{attribute addProperty BoxType "EL5101-0000-0001"}
{attribute addProperty Id "StatusAT %I*USINT811ValueAT %I*UINT1622LatchAT %I*UINT1623"}
{attribute addProperty CRC "1865938148"}
{attribute addProperty SizeInBites "40"}
{attribute addProperty SizeInBytes "5"}
TYPE Inputs_6F37F4E4 :
STRUCT
	{attribute addProperty Name "Status"}
	Status AT %I* : USINT;
	{attribute addProperty Name "Value"}
	Value AT %I* : UINT;
	{attribute addProperty Name "Latch"}
	Latch AT %I* : UINT;
END_STRUCT
END_TYPE

(* stored: Version 1.2.0.0, ProductVersion 3.1.4024.9
   DUT Inputs_6F37F4E4: Id {a34023c1-93ad-4f1b-9b1f-903603b46ba9} *)
